// TwinCAT 3 PLC project HomePLC_LinkManager
// Title: HomePLC Link Manager
// Company: Tom Oyen
// Author: Tom Oyen
// ProjectVersion: 1.0.3
// Description: Link manager
// ProgramVersion: 3.1.4024.0
// libraries:
//   HomePLC DIO, * (Tom Oyen)
//   HomePLC Logging, * (Tom Oyen)
//   Tc2_Standard, * (Beckhoff Automation GmbH)
//   Tc2_System, * (Beckhoff Automation GmbH)
//   Tc3_Module, * (Beckhoff Automation GmbH)
// project tree:
//   / PlcTask.TcTTO
//   POUs/ FB_LinkManager.TcPOU, I_LinkManager.TcIO
//   POUs/IO group/DUTs/ E_DIGroupMode.TcDUT
//   POUs/IO group/ FB_DIGroup.TcPOU, FB_DOGroup.TcPOU, FB_IOGroup.TcPOU, I_DIGroup.TcIO, I_DOGroup.TcIO
//   POUs/Link/DUTs/ ST_CommandTranslation.TcDUT
//   POUs/Link/ FB_Link.TcPOU, I_Link.TcIO
//   Project Information/ F_GetCompany.TcPOU, F_GetTitle.TcPOU, F_GetVersion.TcPOU
//   Version/ Global_Version.TcGVL

CONFIGURATION HomePLC_LinkManager
    RESOURCE PLC ON TwinCAT3
        TASK PlcTask(INTERVAL := T#10ms, PRIORITY := 20);
    END_RESOURCE
END_CONFIGURATION

// ---- POUs/IO group/DUTs/E_DIGroupMode.TcDUT
{attribute 'qualified_only'}
{attribute 'strict'}
// Mode of combining digital input commands
TYPE E_DIGroupMode :
(
	ModeAND := 0,		// All inputs need to be used to issue the command
	ModeOR	:= 1		// One input is sufficient to issue a command
);
END_TYPE

// ---- POUs/Link/DUTs/ST_CommandTranslation.TcDUT
// Translate input commands to output commands
TYPE ST_CommandTranslation :
STRUCT
	OnShortPress	: E_DOCommand := E_DOCommand.None;	// Output command when input command is short press
	OnLongPress		: E_DOCommand := E_DOCommand.None;	// Output command when input command is long press
	OnDoublePress	: E_DOCommand := E_DOCommand.None;	// Output command when input command is double press
	OnHold			: E_DOCommand := E_DOCommand.None;	// Output command when input command is hold
END_STRUCT
END_TYPE

// ---- Version/Global_Version.TcGVL
{attribute 'TcGenerated'}
{attribute 'no-analysis'}
{attribute 'linkalways'}
// This function has been automatically generated from the project information.
VAR_GLOBAL CONSTANT
	{attribute 'const_non_replaced'}
	stLibVersion_HomePLC_Link_Manager : ST_LibVersion := (iMajor := 1, iMinor := 0, iBuild := 3, iRevision := 0, nFlags := 0, sVersion := '1.0.3');
END_VAR

// ---- POUs/IO group/I_DIGroup.TcIO
INTERFACE I_DIGroup

// Add input to group
METHOD AddInput
VAR_INPUT
	IDI			: I_DigitalIn;		// Interface to digital input
END_VAR
END_METHOD

// Gets the total number of IOs in the group
PROPERTY Count : INT
GET
END_GET
END_PROPERTY

// Determine the command from the inputs in the group
METHOD GetCommand : E_DICommand
END_METHOD

// Get a specific input from the group
METHOD GetInput : I_DigitalIn
VAR_INPUT
	nInputIndex		: INT;		// Input index
END_VAR
END_METHOD

// Set input group mode (default OR)
PROPERTY Mode : E_DIGroupMode
SET
END_SET
END_PROPERTY

END_INTERFACE

// ---- POUs/IO group/I_DOGroup.TcIO
INTERFACE I_DOGroup

// Add indicator to group.
// Indicators are defined separately from outputs. Indicators follow outputs and the link between them is defined in the PLC.
// Regardless of how the output is updated (by the PLC or externally), the indicators follow the outputs. 
METHOD AddIndicator
VAR_INPUT
	IDO			: I_DigitalOut;		// Interface to digital output that needs to be an indicator
END_VAR
END_METHOD

// Add output to group
METHOD AddOutput
VAR_INPUT
	IDO			: I_DigitalOut;		// Interface to digital output
END_VAR
END_METHOD

// Gets the total number of IOs in the group
PROPERTY Count : INT
GET
END_GET
END_PROPERTY

// Get a specific output from the group
METHOD GetOutput : I_DigitalOut
VAR_INPUT
	nOutputIndex		: INT;		// Output index
END_VAR
END_METHOD

// Set the command to the outputs in the group
METHOD SetCommand
VAR_INPUT
	eCommand	: E_DOCommand;
END_VAR
END_METHOD

// Update the indicator values based on the value of the outputs
METHOD UpdateIndicators
END_METHOD

END_INTERFACE

// ---- POUs/I_LinkManager.TcIO
// Link manager interface
INTERFACE I_LinkManager

// Commit link so it can be executed
METHOD CommitLink
END_METHOD

// Returns a link that can be configured and then committed
PROPERTY Link : I_Link
GET
END_GET
END_PROPERTY

END_INTERFACE

// ---- POUs/Link/I_Link.TcIO
INTERFACE I_Link

// Get/set if the link needs to be excluded from the links overview
PROPERTY ExcludeFromOverview : BOOL
GET
END_GET
SET
END_SET
END_PROPERTY

// Group of inputs
PROPERTY InputGroup : I_DIGroup
GET
END_GET
SET
END_SET
END_PROPERTY

// Group of outputs
PROPERTY OutputGroup : I_DOGroup
GET
END_GET
SET
END_SET
END_PROPERTY

// Output reaction
PROPERTY OutputReaction : REFERENCE TO ST_CommandTranslation
GET
END_GET
END_PROPERTY

END_INTERFACE

// ---- POUs/FB_LinkManager.TcPOU
// Link manager
FUNCTION_BLOCK FB_LinkManager IMPLEMENTS I_LinkManager
VAR
	aLinks			: ARRAY [0..nMaxSize - 1] OF FB_Link;	// Array of links
	nSize			: INT;									// Number of links in the array
END_VAR
VAR CONSTANT
	nMaxSize		: INT := 100;							// Maximum number of IOs in a group
END_VAR

// Commit link so it can be executed
METHOD CommitLink
IF nSize < nMaxSize THEN
	nSize := nSize + 1;
END_IF
END_METHOD

// Execute links
METHOD Execute
VAR
	i		: INT;		// Iterator variable
END_VAR
// Execute all links
FOR i := 0 TO nSize - 1 DO
	aLinks[i].Execute();
END_FOR
END_METHOD

METHOD GetLink : I_Link
VAR_INPUT
	nIndex		: INT;		// Link index
END_VAR
GetLink := aLinks[nIndex];
END_METHOD

// Returns a link that can be configured and then committed
PROPERTY Link : I_Link
GET
Link := aLinks[nSize];
END_GET
END_PROPERTY

END_FUNCTION_BLOCK

// ---- POUs/Link/FB_Link.TcPOU
// Link between an input and an output group
FUNCTION_BLOCK FB_Link IMPLEMENTS I_Link
VAR
	IInputGroup				: I_DIGroup;				// Input group interface
	IOutputGroup			: I_DOGroup;				// Output group interface
	
	fbInputGroup			: FB_DIGroup;				// Input group FB, in case interface is not set to an FB
	fbOutputGroup			: FB_DOGroup;				// Output group FB, in case interface is not set to an FB
	
	stCommandTranslation	: ST_CommandTranslation;	// Input command to output command translation
	bExcludeFromOverview	: BOOL;						// Set to true to exclude this link from the links overview
END_VAR

// Get/set if the link needs to be excluded from the links overview
PROPERTY ExcludeFromOverview : BOOL
GET
ExcludeFromOverview := bExcludeFromOverview;
END_GET
SET
bExcludeFromOverview := ExcludeFromOverview;
END_SET
END_PROPERTY

// Pass the command from the input group to the output group
METHOD Execute
// Get input command and translate it to an output command
CASE IInputGroup.GetCommand() OF
	E_DICommand.None:
		IOutputGroup.SetCommand(E_DOCommand.None);
	E_DICommand.ShortPress:
		IOutputGroup.SetCommand(stCommandTranslation.OnShortPress);
	E_DICommand.DoublePress:
		IOutputGroup.SetCommand(stCommandTranslation.OnDoublePress);
	E_DICommand.LongPress:
		IOutputGroup.SetCommand(stCommandTranslation.OnLongPress);
	E_DICommand.Hold:
		IOutputGroup.SetCommand(stCommandTranslation.OnHold);
END_CASE

// Update output group indicators
IOutputGroup.UpdateIndicators();

// Do not call the execute method of all IO groups here
// A digital in/output may appear in multiple links and the execute method should not be called more than once per PLC cycle
END_METHOD

METHOD FB_init : BOOL
VAR_INPUT
	bInitRetains : BOOL; // if TRUE, the retain variables are initialized (warm start / cold start)
	bInCopyCode : BOOL;  // if TRUE, the instance afterwards gets moved into the copy code (online change)
END_VAR
// Initialize interfaces with local FBs, can be replaced afterwards if needed
IInputGroup := fbInputGroup;
IOutputGroup := fbOutputGroup;
END_METHOD

// Group of inputs
PROPERTY InputGroup : I_DIGroup
GET
InputGroup := IInputGroup;
END_GET
SET
IInputGroup := InputGroup;
END_SET
END_PROPERTY

// Group of outputs
PROPERTY OutputGroup : I_DOGroup
GET
OutputGroup := IOutputGroup;
END_GET
SET
IOutputGroup := OutputGroup;
END_SET
END_PROPERTY

// Output reaction
PROPERTY OutputReaction : REFERENCE TO ST_CommandTranslation
GET
OutputReaction REF= stCommandTranslation;
END_GET
END_PROPERTY

END_FUNCTION_BLOCK

// ---- POUs/IO group/FB_DIGroup.TcPOU
// Digital input group
FUNCTION_BLOCK FB_DIGroup EXTENDS FB_IOGroup IMPLEMENTS I_DIGroup
VAR
	aIn				: ARRAY [0..nMaxSize - 1] OF I_DigitalIn;	// Array of interfaces of digital inputs
	eMode			: E_DIGroupMode := E_DIGroupMode.ModeOR;	// Command mode of inputs in group (default = OR)
END_VAR

// Add input to group
METHOD AddInput
VAR_INPUT
	IDI			: I_DigitalIn;		// Interface to digital input
END_VAR
IF nSize < nMaxSize THEN
	aIn[nSize] := IDI;
	nSize := nSize + 1;
END_IF
END_METHOD

// Runs the execute method of all digital input FBs in the group.
// Make sure all digital output execute methods are called only once per PLC cyle
METHOD Execute
VAR
	i		: INT;		// Iterator variable
END_VAR
// Call the execute method of all digital inputs in the group
FOR i := 0 TO nSize - 1 DO
	aIn[i].Execute();
END_FOR
END_METHOD

// Determine the command from the inputs in the group
METHOD GetCommand : E_DICommand
VAR
	i				: INT;
	nActive			: INT;
	eCommand		: E_DICommand;
	sTemp			: STRING;
END_VAR
VAR_INST
	eState			: E_DIState;
END_VAR
// Check at least one input is available
IF nSize > 0 THEN
	CASE eMode OF
	E_DIGroupMode.ModeOR:
		// Get command
		eCommand := E_DICommand.None;
		
		FOR i := 0 TO nSize - 1 DO
			// Find first command different from None
			IF aIn[i].Command <> E_DICommand.None THEN
				IF eCommand = E_DICommand.None THEN
					eCommand := aIn[i].Command;
					
					sTemp := 'OR command ';
					sTemp := CONCAT(sTemp, TO_STRING(eCommand));
					fbLogger.AddDebug(sTemp);
				END_IF
			END_IF
		END_FOR
		
		// Issue command
		GetCommand := eCommand;
		
	E_DIGroupMode.ModeAND:
		// Check states
		// Multiple buttons must have been active at the same time with the same state
		nActive := 0;
		FOR i := 0 TO nSize - 1 DO
			IF aIn[i].State <> E_DIState.Idle THEN
				IF eState = E_DIState.Idle THEN
					eState := aIn[i].State;
				END_IF
				IF aIn[i].State = eState THEN
					nActive := nActive + 1;
				END_IF
			END_IF
		END_FOR
		
		// Reset if all inactive
		IF nActive = 0 THEN
			eState := E_DIState.Idle;
		END_IF
		
		// Get command
		eCommand := E_DICommand.None;
		FOR i := 0 TO nSize - 1 DO
			// Find first command different from None
			IF aIn[i].Command <> E_DICommand.None THEN
				IF eCommand = E_DICommand.None THEN
					eCommand := aIn[i].Command;
				END_IF
			END_IF
		END_FOR
		
		IF eCommand <> E_DICommand.None THEN
			// All commands need to be the same
			// Assume command matches detected states
			IF nActive = nSize THEN
				GetCommand := eCommand;
				
				sTemp := 'AND command ';
				sTemp := CONCAT(sTemp, TO_STRING(eCommand));
				sTemp := CONCAT(sTemp, ' by ');
				sTemp := CONCAT(sTemp, INT_TO_STRING(nActive));
				sTemp := CONCAT(sTemp, ' inputs');
				fbLogger.AddDebug(sTemp);
			END_IF
		ELSE
			GetCommand := E_DICommand.None;
		END_IF
	END_CASE
ELSE
	GetCommand := E_DICommand.None;
END_IF
END_METHOD

// Get a specific input from the group
METHOD GetInput : I_DigitalIn
VAR_INPUT
	nInputIndex		: INT;		// Input index
END_VAR
GetInput := aIn[nInputIndex];
END_METHOD

// Set input group mode (default OR)
PROPERTY Mode : E_DIGroupMode
SET
eMode := Mode;
END_SET
END_PROPERTY

END_FUNCTION_BLOCK

// ---- POUs/IO group/FB_IOGroup.TcPOU
{attribute 'reflection'} 
FUNCTION_BLOCK FB_IOGroup
VAR
	nSize			: INT;			// Number of IOs in this group
	
	fbLogger		: class_Tc3EventLogger;
	
	// Use attributes to copy instance name to sName
	{attribute 'instance-path'} 
    {attribute 'noinit'} 
    sName			: STRING; 		// Instance name
END_VAR
VAR CONSTANT
	nMaxSize		: INT := 100;	// Maximum number of IOs in a group
END_VAR

// Gets the total number of IOs in the group
PROPERTY Count : INT
GET
Count := nSize;
END_GET
END_PROPERTY

METHOD FB_init : BOOL
VAR_INPUT
	bInitRetains : BOOL; // if TRUE, the retain variables are initialized (warm start / cold start)
	bInCopyCode : BOOL;  // if TRUE, the instance afterwards gets moved into the copy code (online change)
END_VAR
fbLogger.Init(sSource := sName, bEnableVerbose := FALSE);
END_METHOD

END_FUNCTION_BLOCK

// ---- POUs/IO group/FB_DOGroup.TcPOU
// Digital output group
FUNCTION_BLOCK FB_DOGroup EXTENDS FB_IOGroup IMPLEMENTS I_DOGroup
VAR
	aOut			: ARRAY [0..nMaxSize - 1] OF I_DigitalOut;		// Array of interfaces to digital outputs
	
	aIndicator		: ARRAY [0..nMaxSize - 1] OF I_DigitalOut;		// Array of interfaces to digital outputs that serve as indicators
	nSizeIndicators	: INT;											// Size of indicator array
END_VAR

// Add indicator to group.
// Indicators are defined separately from outputs. Indicators follow outputs and the link between them is defined in the PLC.
// Regardless of how the output is updated (by the PLC or externally), the indicators follow the outputs. 
METHOD AddIndicator
VAR_INPUT
	IDO			: I_DigitalOut;		// Interface to digital output that needs to be an indicator
END_VAR
IF nSizeIndicators < nMaxSize THEN
	aIndicator[nSizeIndicators] := IDO;
	nSizeIndicators := nSizeIndicators + 1;
END_IF
END_METHOD

// Add output to group
METHOD AddOutput
VAR_INPUT
	IDO			: I_DigitalOut;		// Interface to digital output
END_VAR
IF nSize < nMaxSize THEN
	aOut[nSize] := IDO;
	nSize := nSize + 1;
END_IF
END_METHOD

// Runs the execute method of all digital output FBs in the group.
// Make sure all digital output execute methods are called only once per PLC cyle
METHOD Execute
VAR
	i		: INT;		// Iterator variable
END_VAR
// Call the execute method of all digital outputs in the group
FOR i := 0 TO nSize - 1 DO
	aOut[i].Execute();
END_FOR
END_METHOD

// Get a specific output from the group
METHOD GetOutput : I_DigitalOut
VAR_INPUT
	nOutputIndex		: INT;		// Output index
END_VAR
GetOutput := aOut[nOutputIndex];
END_METHOD

// Set the command to the outputs in the group
METHOD SetCommand
VAR_INPUT
	eCommand	: E_DOCommand;
END_VAR
VAR
	i			: INT;
END_VAR
FOR i := 0 TO nSize - 1 DO
	IF aOut[i].Command = E_DOCommand.None THEN
		// No command yet, set new command
		aOut[i].SetCommand(eCommand);
	ELSE
		// A command was already issued
		// Do nothing
	END_IF
END_FOR
END_METHOD

// Update the indicator values based on the value of the outputs
METHOD UpdateIndicators
VAR
	i		: INT;		// Iterator variable
	bOn		: BOOL;		// True if at least one output is on
END_VAR
// Check if there is at least one output in the group since at least one output is needed to determine the output value
IF nSize > 0 THEN
	// Check if at least one output is on
	// If only the PLC manipulates the output group all outputs will have the same value
	// However, if a single output is manipulated externally (by ADS) one output can have a different value
	// In this case, OR the output values and turn on the indicator if at least one output is on
	bOn := FALSE;
	FOR i := 0 TO nSize - 1 DO
		bOn := bOn OR aOut[i].Output;
	END_FOR
	
	// Set output value of all indicators to that of the value of the output group
	FOR i := 0 TO nSizeIndicators - 1 DO
		aIndicator[i].Output := bOn;
	END_FOR
END_IF
END_METHOD

END_FUNCTION_BLOCK

// ---- Project Information/F_GetCompany.TcPOU
// This function has been automatically generated from the project information.
{attribute 'signature_flag' := '1073741824'}
{attribute 'TcGenerated'}
{attribute 'no-analysis'}
FUNCTION F_GetCompany : WSTRING
VAR_INPUT
	
END_VAR

F_GetCompany := "Tom Oyen";

END_FUNCTION

// ---- Project Information/F_GetTitle.TcPOU
// This function has been automatically generated from the project information.
{attribute 'signature_flag' := '1073741824'}
{attribute 'TcGenerated'}
{attribute 'no-analysis'}
FUNCTION F_GetTitle : WSTRING
VAR_INPUT
	
END_VAR

F_GetTitle := "HomePLC Link Manager";

END_FUNCTION

// ---- Project Information/F_GetVersion.TcPOU
// This function has been automatically generated from the project information.
{attribute 'signature_flag' := '1073741824'}
{attribute 'TcGenerated'}
{attribute 'no-analysis'}
FUNCTION F_GetVersion : ST_LibVersion
VAR_INPUT
	
END_VAR

F_GetVersion.iMajor := 1;
F_GetVersion.iMinor := 0;
F_GetVersion.iBuild := 3;
F_GetVersion.iRevision := 0;
F_GetVersion.sVersion := '1.0.3';
F_GetVersion.nFlags := 0;

END_FUNCTION
